{attribute 'GeneratedUsingTerminal: EL5001-0011-0019'}
{attribute addProperty BoxType "EL5001-0011-0019"}
{attribute addProperty Id "SSI_InputsAT %I*SSI_Inputs_8BC18DAC9WcStateAT %I*WcState_9091E0EB2InfoDataAT %I*InfoData_1088C70510"}
{attribute addProperty CRC "3084537757"}
{attribute addProperty Size "21"}
TYPE EL5001_B7DA4F9D EXTENDS EtcSlaveTerminalBase_947E5A46 :
STRUCT
	{attribute addProperty Name "SSI_Inputs"}
	SSI_Inputs : SSI_Inputs_8BC18DAC;
	{attribute addProperty Name "WcState"}
	WcState : WcState_9091E0EB;
	{attribute addProperty Name "InfoData"}
	InfoData : InfoData_1088C705;
END_STRUCT
END_TYPE

(* stored: Version 1.2.0.0, ProductVersion 3.1.4024.9
   DUT EL5001_B7DA4F9D: Id {8d3fdefc-76fe-41aa-8930-694c88b486cf} *)
